// TIA Portal V18 export
// export: Created 2026-03-12T16:04:35.55371Z, ExportSetting WithDefaults, DisplayName Totally Integrated Automation Portal, DisplayVersion V18 Update 5, DisplayName TIA Portal Openness, DisplayVersion V18 Update 5, DisplayName TIA Portal Version Control Interface, DisplayVersion V18, DisplayName SINAMICS Startdrive Advanced, DisplayVersion V18, DisplayName SINAMICS Startdrive G130, G150, S120, S150, SINAMICS MV, S210, DisplayVersion V18, DisplayName SINAMICS Startdrive G110M, G120, G120C, G120D, G120P, G115D, DisplayVersion V18, DisplayName STEP 7 Professional, DisplayVersion V18 Update 5, DisplayName STEP 7 Safety, DisplayVersion V18, DisplayName WinCC Professional, DisplayVersion V18 Update 5
FUNCTION_BLOCK "FB MODBUS MASTER BLOCK MMW"   // FB18, LAD
{ S7_Optimized_Access := 'TRUE' }
VERSION : 0.1
// Instanciamento do Bloco Modbus Master para cada Driver (Multimedidor)
// 
// Network 1: Chamada por índice de endereço
// Network 2: Falha de comunicação Modbus
// Network 3: Reset do módulo de comunicação Modbus
// stored: AutoNumber true, IsIECCheckEnabled false, IsRetainMemResEnabled false, MemoryReserve 100, SetENOAutomatically false, UDAEnableTagReadback false
   VAR_INPUT
      INDEX_DRIVER : Int;   // Índice do driver, numerando a instância de cada um
      INDEX_ADDR : Int;   // Índice do endereço, numerando a ordem de leitura de cada um
      TRIGGER : Bool;   // Gatilho de chamada do bloco. (Recebido da instância do FB SCAN DRIVERS conforme o DONE do bloco master)
      MODBUS_ID : Int;   // Endereço ID do Modbus
      ARRAY_ADDR_MMW : Array[0..40] of Int;   // Array de endereços (Todos os 41 endereços cadastrados na tabela Modbus do equipamento)
      INDEX_BLOCK : Int;   // Índice de instância, para definir quando os blocos Master serão chamados
      CICLE_TIMES_SET_ALARME : Int;   // Cadastro do "Tryout", número de tentativas de comunicação antes de acionar o erro
   END_VAR
   VAR_OUTPUT
      DRIVER_ERROR_COMUNIC : Bool;   // Erro de comunicação Modbus
      ERROR_CODE : Word;   // Código do erro de comunicação Modbus
      RESET_PTP : Bool;   // Saída para reset do módulo Commload
   END_VAR
   VAR_IN_OUT
      MODBUS_MASTER : Modbus_Master;
      ARRAY_MMW : Array[0..40] of Real;   // Array da DB GLOBAL onde os registros são armazenados
   END_VAR
   VAR
      PULSE_SCAN { S7_SetPoint := 'True'} : Bool;   // Pulso para contagem do número de tentativas de comunicação mal sucedidas
      COUT_PULSE : Bool;   // Memória auxiliar do pulso
      ERROR_CICLES : Int;   // Memória de incremento a cada pulso do PULSE_SCAN
      ACTUAL_ERROR : Word;   // Captura do código de erro na tentativa de comunicação mal sucedida
      MASTER_DRIVER_LAST_ERROR : Int;   // Índice do driver que registrou o último erro
      ARRAY_READ_MMW : Array[0..40] of Real;   // Array local para armazenar temporariamente as leituras antes de mover à DB GLOBAL
      HABILITA_RESET : Bool;   // Habilita reset após intervalo de tempo
      AUX_RESET : Bool;   // Memória auxiliar para o reset modbus
      RESET_TIMER_1 : IEC_TIMER;   // Tempo de cooldown para utilizar o reset novamente
      RESET_TIMER_2 : IEC_TIMER;   // Tempo de saída acionada (reset)
   END_VAR
   VAR_TEMP   // added for the SCL form of the ladder/FBD networks
      _w1 : Bool;
      _w2 : Bool;
   END_VAR
BEGIN

REGION Network 1: Function BLock MODBUS MASTER BLOCK MMW
   // Ao chamar o bloco, o índice de endereço irá alternar entre os 41 endereços do multimedidor. Essas informações são registradas em um array de tamanho 41 e movidos à DB GLOBAL.
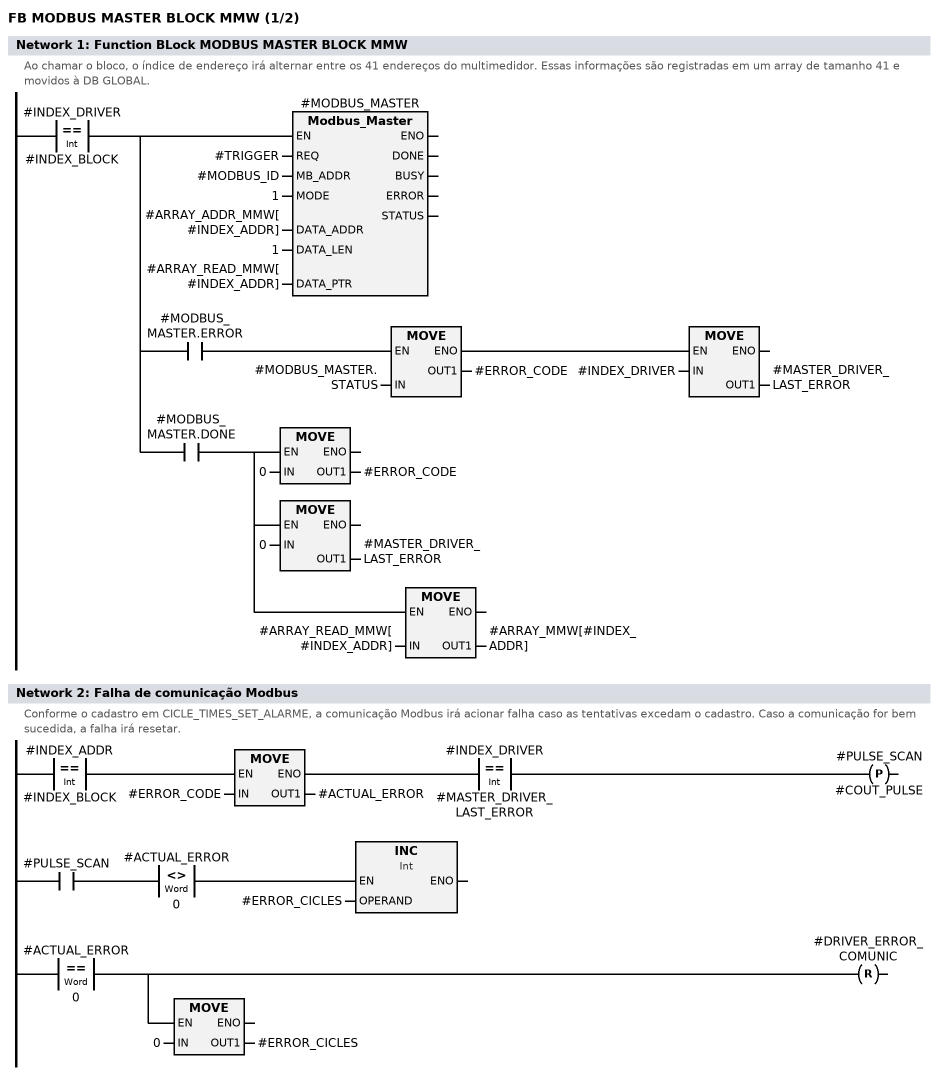
   RUNG wire#powerrail
      { S7_Templates := "SrcType := Int" } EQ_Contact(in1 := #INDEX_DRIVER, in2 := #INDEX_BLOCK)
      wire#w1
      #MODBUS_MASTER.Modbus_Master(REQ := #TRIGGER, MB_ADDR := #MODBUS_ID, MODE := 1, DATA_ADDR := #ARRAY_ADDR_MMW[#INDEX_ADDR], DATA_LEN := 1, DATA_PTR := #ARRAY_READ_MMW[#INDEX_ADDR], DONE =>, BUSY =>, ERROR =>, STATUS =>)
   END_RUNG
   RUNG wire#w1
      Contact( #MODBUS_MASTER.ERROR )
      Move(in := #MODBUS_MASTER.STATUS, out1 => #ERROR_CODE)
      Move(in := #INDEX_DRIVER, out1 => #MASTER_DRIVER_LAST_ERROR)
   END_RUNG
   RUNG wire#w1
      Contact( #MODBUS_MASTER.DONE )
      wire#w2
      Move(in := 0, out1 => #ERROR_CODE)
   END_RUNG
   RUNG wire#w2
      Move(in := 0, out1 => #MASTER_DRIVER_LAST_ERROR)
   END_RUNG
   RUNG wire#w2
      Move(in := #ARRAY_READ_MMW[#INDEX_ADDR], out1 => #ARRAY_MMW[#INDEX_ADDR])
   END_RUNG
   // the same network as SCL:
   #_w1 := #INDEX_DRIVER = #INDEX_BLOCK;
   IF #_w1 THEN
       #MODBUS_MASTER(REQ := #TRIGGER,   // Modbus_Master
                      MB_ADDR := #MODBUS_ID,
                      MODE := 1,
                      DATA_ADDR := #ARRAY_ADDR_MMW[#INDEX_ADDR],
                      DATA_LEN := 1,
                      DATA_PTR := #ARRAY_READ_MMW[#INDEX_ADDR]);
   END_IF;
   IF #_w1 AND #MODBUS_MASTER.ERROR THEN
       #ERROR_CODE := #MODBUS_MASTER.STATUS;
       #MASTER_DRIVER_LAST_ERROR := #INDEX_DRIVER;
   END_IF;
   IF #_w1 AND #MODBUS_MASTER.DONE THEN
       #ERROR_CODE := 0;
       #MASTER_DRIVER_LAST_ERROR := 0;
       #ARRAY_MMW[#INDEX_ADDR] := #ARRAY_READ_MMW[#INDEX_ADDR];
   END_IF;
END_REGION

REGION Network 2: Falha de comunicação Modbus
   // Conforme o cadastro em CICLE_TIMES_SET_ALARME, a comunicação Modbus irá acionar falha caso as tentativas excedam o cadastro. Caso a comunicação for bem sucedida, a falha irá resetar.
   #_w1 := #INDEX_ADDR = #INDEX_BLOCK;
   IF #_w1 THEN #ACTUAL_ERROR := #ERROR_CODE; END_IF;
   #_w2 := #_w1 AND (#INDEX_DRIVER = #MASTER_DRIVER_LAST_ERROR);
   #PULSE_SCAN := #_w2 AND NOT #COUT_PULSE;   // rising edge
   #COUT_PULSE := #_w2;
   IF #PULSE_SCAN AND (#ACTUAL_ERROR <> 0) THEN #ERROR_CICLES := #ERROR_CICLES + 1; END_IF;
   IF #ACTUAL_ERROR = 0 THEN
       #DRIVER_ERROR_COMUNIC := FALSE;
       #ERROR_CICLES := 0;
   END_IF;
END_REGION

REGION Network 3: Reset do módulo de comunicação Modbus
   // Reset ao identificar erro de comunicação.
   // Tempo de cooldown 600s (10min): Intervalo de tempo após o reset para resetar novamente caso o equipamento ainda esteja em erro.
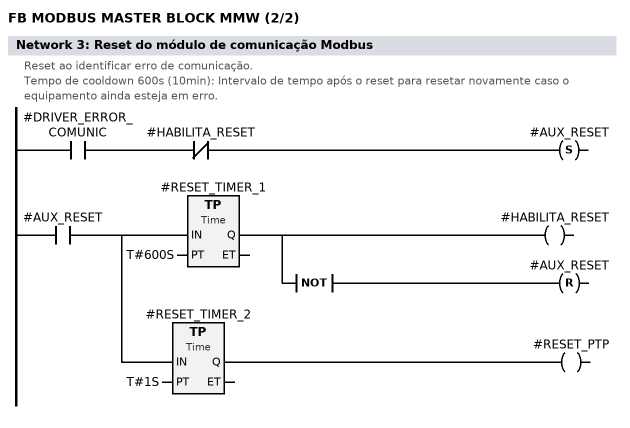
   RUNG wire#powerrail
      Contact( #DRIVER_ERROR_COMUNIC )
      I_Contact( #HABILITA_RESET )
      S_Coil( #AUX_RESET )
   END_RUNG
   RUNG wire#powerrail
      Contact( #AUX_RESET )
      wire#w1
      { S7_Templates := "time_type := Time" } #RESET_TIMER_1.TP(pt := T#600S, et =>)
      wire#w2
      Coil( #HABILITA_RESET )
   END_RUNG
   RUNG wire#w2
      Not()
      R_Coil( #AUX_RESET )
   END_RUNG
   RUNG wire#w1
      { S7_Templates := "time_type := Time" } #RESET_TIMER_2.TP(pt := T#1S, et =>)
      Coil( #RESET_PTP )
   END_RUNG
   // the same network as SCL:
   IF #DRIVER_ERROR_COMUNIC AND NOT #HABILITA_RESET THEN #AUX_RESET := TRUE; END_IF;
   #RESET_TIMER_1.TP(IN := #AUX_RESET, PT := T#600S);
   #HABILITA_RESET := #RESET_TIMER_1.Q;
   #_w1 := #AUX_RESET;
   IF NOT #RESET_TIMER_1.Q THEN #AUX_RESET := FALSE; END_IF;
   #RESET_TIMER_2.TP(IN := #_w1, PT := T#1S);
   #RESET_PTP := #RESET_TIMER_2.Q;
END_REGION
END_FUNCTION_BLOCK
